Universal Robots PolyScope program: test.urp

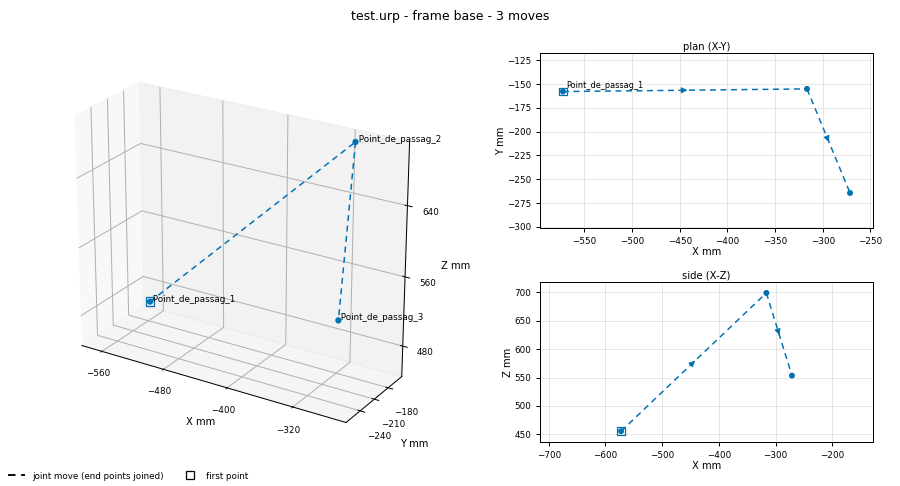
[picture p0: tool path of test.urp in frame base, 3 of 3 moves have a stored position in this frame; points joined in program order, loops and branches not executed]
ProgramRoot directory=/programs; kinematics=(a=[0, -0.425, -0.39225, 0, 0, 0], d=[0.08916, 0, 0, 0.10915, 0.09465, 0.0823], alpha=[1.5708, 0, 0, 1.5708, -1.5708, 0], deltaTheta=[0, 0, 0, 0, 0, 0], status=notInitialized); name=test; programVersion=(project__name=PolyScope, major__version=1, minor__version=6, svn__revision=9671, build__date=Dec 17 2012, 15:17:18); robotEnvironmentFileName=default
  MainProgram cartesianAcceleration=1.2; cartesianSpeed=0.25; jointAcceleration=1.3962634015954636; jointSpeed=1.0471975511965976; moveAsFastAsPossible=true; sharedProcessMoveBlendRadius=0.025; featureReference=(installationNameReference=Base); motionType=JOINT_SPACE
    Move cartesianAcceleration=1.2; cartesianSpeed=0.25; jointAcceleration=25.0; jointSpeed=3.2; moveAsFastAsPossible=true; sharedProcessMoveBlendRadius=0.025; featureReference=(installationNameReference=Base); motionType=JOINT_SPACE
      Waypoint blendRadius=0.05; cartesianAcceleration=1.2; cartesianSpeed=0.25; jointAcceleration=1.3962634015954636; jointSpeed=1.0471975511965976; nextMotionTime=2.0; stoppoint=true; useSharedBlendParameter=true; useSharedParameters=true; position=TCP in base x=-572.558 y=-157.902 z=455.473 mm, rx=-1.3805 ry=-2.7909 rz=0.3122 rad; joints [3.483, -78.283, 75.312, -93.394, -80.436, -33.345] deg; positionType=FIXED_POSITION; waypointPoseInFeatureCoordinates=(pos=(x=-0.5725584099112776, y=-0.15790197754161467, z=0.45547308102914896), rot=(x=-1.3805005261660428, y=-2.790856599438613, z=0.31215938031251783)); name=Point_de_passag_1
      Wait analogComparison=0; analogInputRange=0; analogValue=0.0; digitalValue=0; selectedAnalogSensor=-1; selectedDigitalSensor=-1; waitTime=0.5; type=TIMER_WAIT
      Waypoint blendRadius=0.05; cartesianAcceleration=1.2; cartesianSpeed=0.25; jointAcceleration=1.3962634015954636; jointSpeed=1.0471975511965976; nextMotionTime=2.0; stoppoint=true; useSharedBlendParameter=true; useSharedParameters=true; position=TCP in base x=-316.5 y=-155.144 z=699.131 mm, rx=-1.0593 ry=-2.3905 rz=0.63 rad; joints [5.721, -106.886, 74.033, -93.393, -80.436, -33.345] deg; positionType=FIXED_POSITION; waypointPoseInFeatureCoordinates=(pos=(x=-0.3164997237606843, y=-0.15514437775641943, z=0.6991311621166452), rot=(x=-1.0592515468081807, y=-2.3904605502071563, z=0.6300121260779334)); name=Point_de_passag_2
      Waypoint blendRadius=0.05; cartesianAcceleration=1.2; cartesianSpeed=0.25; jointAcceleration=1.3962634015954636; jointSpeed=1.0471975511965976; nextMotionTime=2.0; specifyNextMotionTime=true; stoppoint=true; useSharedBlendParameter=true; useSharedParameters=true; position=TCP in base x=-271.379 y=-264.306 z=553.399 mm, rx=-0.704 ry=-2.723 rz=0.6163 rad; joints [25.511, -109.805, 96.155, -103.973, -81.258, -33.345] deg; positionType=FIXED_POSITION; waypointPoseInFeatureCoordinates=(pos=(x=-0.27137912219963756, y=-0.2643058669130448, z=0.5533987928577502), rot=(x=-0.7039940880223955, y=-2.723017619770039, z=0.6162999224501475)); name=Point_de_passag_3
